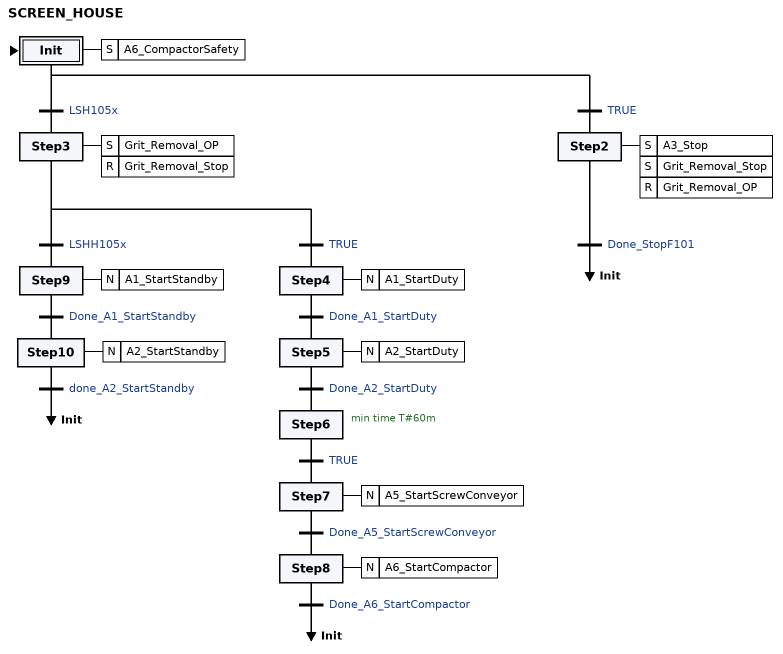
[picture p48: SCREEN_HOUSE (SFC)]
INITIAL_STEP Init:
	A6_CompactorSafety(S);
END_STEP
TRANSITION FROM Init TO Step3 := LSH105x;
END_TRANSITION
TRANSITION FROM Init TO Step2 := TRUE;
END_TRANSITION
STEP Step3:
	Grit_Removal_OP(S);
	Grit_Removal_Stop(R);
END_STEP
TRANSITION FROM Step3 TO Step9 := LSHH105x;
END_TRANSITION
TRANSITION FROM Step3 TO Step4 := TRUE;
END_TRANSITION
STEP Step9:
	A1_StartStandby(N);
END_STEP
TRANSITION FROM Step9 TO Step10 := Done_A1_StartStandby;
END_TRANSITION
STEP Step10:
	A2_StartStandby(N);
END_STEP
TRANSITION FROM Step10 TO Init := done_A2_StartStandby;
END_TRANSITION
STEP Step4:
	A1_StartDuty(N);
END_STEP
TRANSITION FROM Step4 TO Step5 := Done_A1_StartDuty;
END_TRANSITION
STEP Step5:
	A2_StartDuty(N);
END_STEP
TRANSITION FROM Step5 TO Step6 := Done_A2_StartDuty;
END_TRANSITION
STEP Step6: (* min time T#60m *)
END_STEP
TRANSITION FROM Step6 TO Step7 := TRUE;
END_TRANSITION
STEP Step7:
	A5_StartScrewConveyor(N);
END_STEP
TRANSITION FROM Step7 TO Step8 := Done_A5_StartScrewConveyor;
END_TRANSITION
STEP Step8:
	A6_StartCompactor(N);
END_STEP
TRANSITION FROM Step8 TO Init := Done_A6_StartCompactor;
END_TRANSITION
STEP Step2:
	A3_Stop(S);
	Grit_Removal_Stop(S);
	Grit_Removal_OP(R);
END_STEP
TRANSITION FROM Step2 TO Init := Done_StopF101;
END_TRANSITION
END_FUNCTION_BLOCK
ACTION A1_StartDuty:
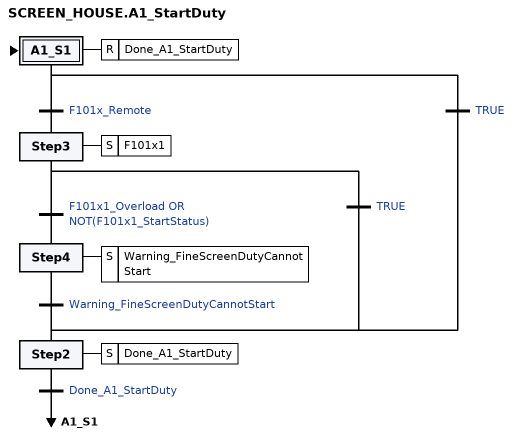
INITIAL_STEP A1_S1:
	Done_A1_StartDuty(R);
END_STEP
TRANSITION FROM A1_S1 TO Step3 := F101x_Remote;
END_TRANSITION
TRANSITION FROM A1_S1 TO Step2 := TRUE;
END_TRANSITION
STEP Step3:
	F101x1(S);
END_STEP
TRANSITION FROM Step3 TO Step4 := F101x1_Overload OR NOT(F101x1_StartStatus);
END_TRANSITION
TRANSITION FROM Step3 TO Step2 := TRUE;
END_TRANSITION
STEP Step4:
	Warning_FineScreenDutyCannotStart(S);
END_STEP
TRANSITION FROM Step4 TO Step2 := Warning_FineScreenDutyCannotStart;
END_TRANSITION
STEP Step2:
	Done_A1_StartDuty(S);
END_STEP
TRANSITION FROM Step2 TO A1_S1 := Done_A1_StartDuty;
END_TRANSITION
END_ACTION
ACTION A1_StartStandby:
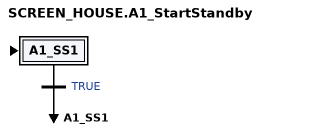
INITIAL_STEP A1_SS1:
END_STEP
TRANSITION FROM A1_SS1 TO A1_SS1 := TRUE;
END_TRANSITION
END_ACTION
ACTION A1_StopDuty:
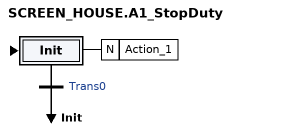
INITIAL_STEP Init:
	Action_1(N);
END_STEP
TRANSITION FROM Init TO Init := Trans0;
END_TRANSITION
END_ACTION
ACTION A1_StopStandby:
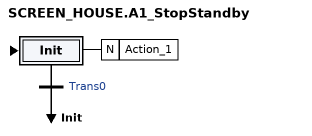
INITIAL_STEP Init:
	Action_1(N);
END_STEP
TRANSITION FROM Init TO Init := Trans0;
END_TRANSITION
END_ACTION
ACTION A2_StartDuty:
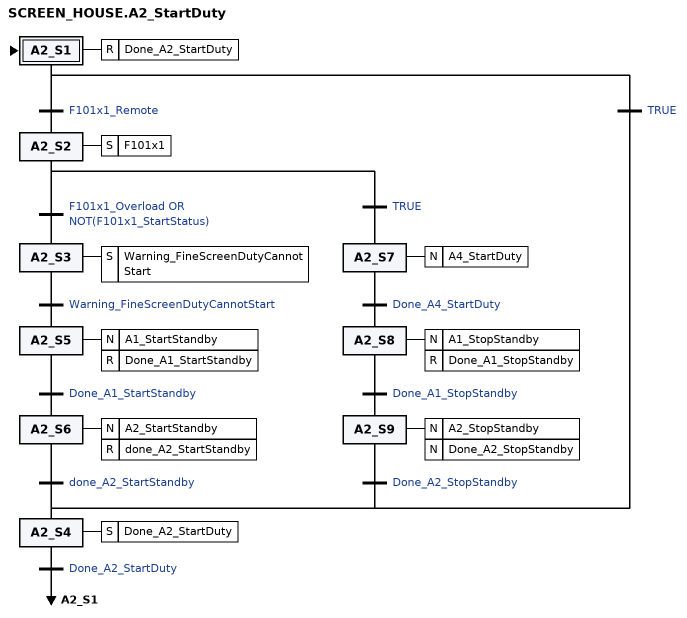
INITIAL_STEP A2_S1:
	Done_A2_StartDuty(R);
END_STEP
TRANSITION FROM A2_S1 TO A2_S2 := F101x1_Remote;
END_TRANSITION
TRANSITION FROM A2_S1 TO A2_S4 := TRUE;
END_TRANSITION
STEP A2_S2:
	F101x1(S);
END_STEP
TRANSITION FROM A2_S2 TO A2_S3 := F101x1_Overload OR NOT(F101x1_StartStatus);
END_TRANSITION
TRANSITION FROM A2_S2 TO A2_S7 := TRUE;
END_TRANSITION
STEP A2_S3:
	Warning_FineScreenDutyCannotStart(S);
END_STEP
TRANSITION FROM A2_S3 TO A2_S5 := Warning_FineScreenDutyCannotStart;
END_TRANSITION
STEP A2_S5:
	A1_StartStandby(N);
	Done_A1_StartStandby(R);
END_STEP
TRANSITION FROM A2_S5 TO A2_S6 := Done_A1_StartStandby;
END_TRANSITION
STEP A2_S6:
	A2_StartStandby(N);
	done_A2_StartStandby(R);
END_STEP
TRANSITION FROM A2_S6 TO A2_S4 := done_A2_StartStandby;
END_TRANSITION
STEP A2_S7:
	A4_StartDuty(N);
END_STEP
TRANSITION FROM A2_S7 TO A2_S8 := Done_A4_StartDuty;
END_TRANSITION
STEP A2_S8:
	A1_StopStandby(N);
	Done_A1_StopStandby(R);
END_STEP
TRANSITION FROM A2_S8 TO A2_S9 := Done_A1_StopStandby;
END_TRANSITION
STEP A2_S9:
	A2_StopStandby(N);
	Done_A2_StopStandby(N);
END_STEP
TRANSITION FROM A2_S9 TO A2_S4 := Done_A2_StopStandby;
END_TRANSITION
STEP A2_S4:
	Done_A2_StartDuty(S);
END_STEP
TRANSITION FROM A2_S4 TO A2_S1 := Done_A2_StartDuty;
END_TRANSITION
END_ACTION
ACTION A2_StartStandby:
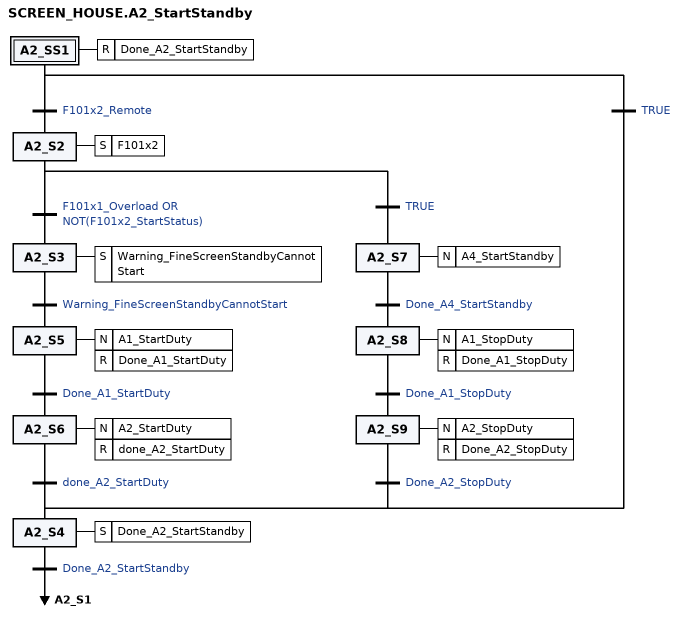
INITIAL_STEP A2_SS1:
	Done_A2_StartStandby(R);
END_STEP
TRANSITION FROM A2_SS1 TO A2_S2 := F101x2_Remote;
END_TRANSITION
TRANSITION FROM A2_SS1 TO A2_S4 := TRUE;
END_TRANSITION
STEP A2_S2:
	F101x2(S);
END_STEP
TRANSITION FROM A2_S2 TO A2_S3 := F101x1_Overload OR NOT(F101x2_StartStatus);
END_TRANSITION
TRANSITION FROM A2_S2 TO A2_S7 := TRUE;
END_TRANSITION
STEP A2_S3:
	Warning_FineScreenStandbyCannotStart(S);
END_STEP
TRANSITION FROM A2_S3 TO A2_S5 := Warning_FineScreenStandbyCannotStart;
END_TRANSITION
STEP A2_S5:
	A1_StartDuty(N);
	Done_A1_StartDuty(R);
END_STEP
TRANSITION FROM A2_S5 TO A2_S6 := Done_A1_StartDuty;
END_TRANSITION
STEP A2_S6:
	A2_StartDuty(N);
	done_A2_StartDuty(R);
END_STEP
TRANSITION FROM A2_S6 TO A2_S4 := done_A2_StartDuty;
END_TRANSITION
STEP A2_S7:
	A4_StartStandby(N);
END_STEP
TRANSITION FROM A2_S7 TO A2_S8 := Done_A4_StartStandby;
END_TRANSITION
STEP A2_S8:
	A1_StopDuty(N);
	Done_A1_StopDuty(R);
END_STEP
TRANSITION FROM A2_S8 TO A2_S9 := Done_A1_StopDuty;
END_TRANSITION
STEP A2_S9:
	A2_StopDuty(N);
	Done_A2_StopDuty(R);
END_STEP
TRANSITION FROM A2_S9 TO A2_S4 := Done_A2_StopDuty;
END_TRANSITION
STEP A2_S4:
	Done_A2_StartStandby(S);
END_STEP
TRANSITION FROM A2_S4 TO A2_S1 := Done_A2_StartStandby;
END_TRANSITION
END_ACTION
ACTION A2_StopDuty:
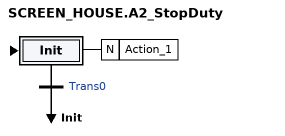
INITIAL_STEP Init:
	Action_1(N);
END_STEP
TRANSITION FROM Init TO Init := Trans0;
END_TRANSITION
END_ACTION
ACTION A2_StopStandby:
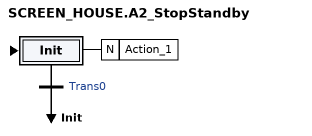
INITIAL_STEP Init:
	Action_1(N);
END_STEP
TRANSITION FROM Init TO Init := Trans0;
END_TRANSITION
END_ACTION
ACTION A3_Stop:
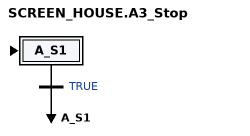
INITIAL_STEP A_S1:
END_STEP
TRANSITION FROM A_S1 TO A_S1 := TRUE;
END_TRANSITION
END_ACTION
ACTION A4_StartDuty:
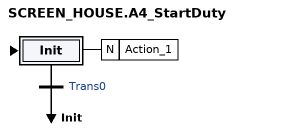
INITIAL_STEP Init:
	Action_1(N);
END_STEP
TRANSITION FROM Init TO Init := Trans0;
END_TRANSITION
END_ACTION
ACTION A4_StartStandby:
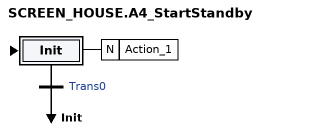
INITIAL_STEP Init:
	Action_1(N);
END_STEP
TRANSITION FROM Init TO Init := Trans0;
END_TRANSITION
END_ACTION
ACTION A5_ResetScrew:
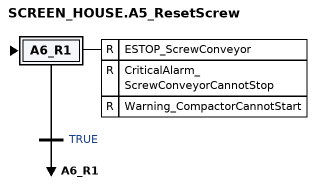
INITIAL_STEP A6_R1:
	ESTOP_ScrewConveyor(R);
	CriticalAlarm_ScrewConveyorCannotStop(R);
	Warning_CompactorCannotStart(R);
END_STEP
TRANSITION FROM A6_R1 TO A6_R1 := TRUE;
END_TRANSITION
END_ACTION
ACTION A5_StartScrewConveyor:
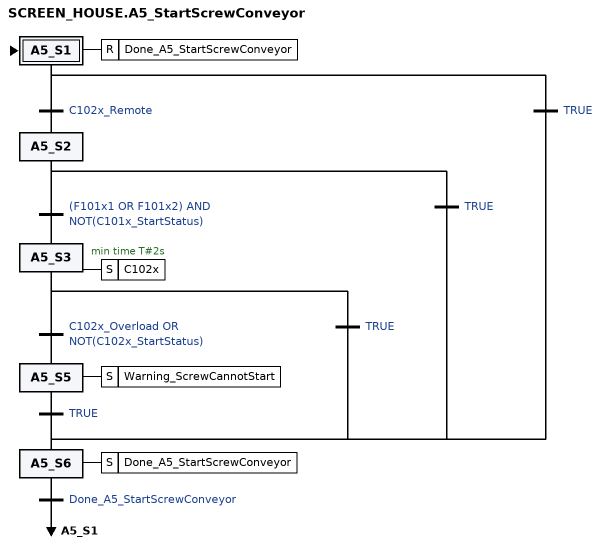
INITIAL_STEP A5_S1:
	Done_A5_StartScrewConveyor(R);
END_STEP
TRANSITION FROM A5_S1 TO A5_S2 := C102x_Remote;
END_TRANSITION
TRANSITION FROM A5_S1 TO A5_S6 := TRUE;
END_TRANSITION
STEP A5_S2:
END_STEP
TRANSITION FROM A5_S2 TO A5_S3 := (F101x1 OR F101x2) AND NOT(C101x_StartStatus);
END_TRANSITION
TRANSITION FROM A5_S2 TO A5_S6 := TRUE;
END_TRANSITION
STEP A5_S3: (* min time T#2s *)
	C102x(S);
END_STEP
TRANSITION FROM A5_S3 TO A5_S5 := C102x_Overload OR NOT(C102x_StartStatus);
END_TRANSITION
TRANSITION FROM A5_S3 TO A5_S6 := TRUE;
END_TRANSITION
STEP A5_S5:
	Warning_ScrewCannotStart(S);
END_STEP
TRANSITION FROM A5_S5 TO A5_S6 := TRUE;
END_TRANSITION
STEP A5_S6:
	Done_A5_StartScrewConveyor(S);
END_STEP
TRANSITION FROM A5_S6 TO A5_S1 := Done_A5_StartScrewConveyor;
END_TRANSITION
END_ACTION
ACTION A5_StopScrewConveyor:
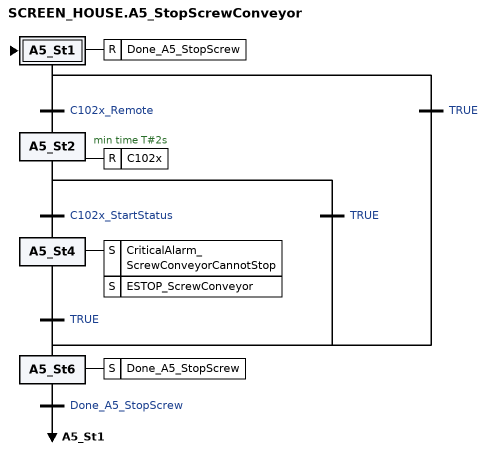
INITIAL_STEP A5_St1:
	Done_A5_StopScrew(R);
END_STEP
TRANSITION FROM A5_St1 TO A5_St2 := C102x_Remote;
END_TRANSITION
TRANSITION FROM A5_St1 TO A5_St6 := TRUE;
END_TRANSITION
STEP A5_St2: (* min time T#2s *)
	C102x(R);
END_STEP
TRANSITION FROM A5_St2 TO A5_St4 := C102x_StartStatus;
END_TRANSITION
TRANSITION FROM A5_St2 TO A5_St6 := TRUE;
END_TRANSITION
STEP A5_St4:
	CriticalAlarm_ScrewConveyorCannotStop(S);
	ESTOP_ScrewConveyor(S);
END_STEP
TRANSITION FROM A5_St4 TO A5_St6 := TRUE;
END_TRANSITION
STEP A5_St6:
	Done_A5_StopScrew(S);
END_STEP
TRANSITION FROM A5_St6 TO A5_St1 := Done_A5_StopScrew;
END_TRANSITION
END_ACTION
ACTION A6_CompactorSafety:
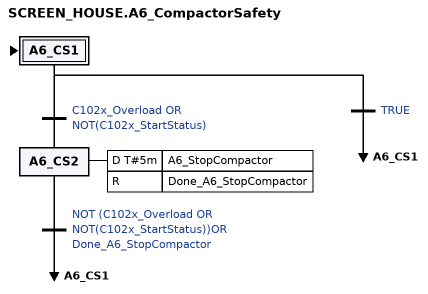
INITIAL_STEP A6_CS1:
END_STEP
TRANSITION FROM A6_CS1 TO A6_CS2 := C102x_Overload OR NOT(C102x_StartStatus);
END_TRANSITION
TRANSITION FROM A6_CS1 TO A6_CS1 := TRUE;
END_TRANSITION
STEP A6_CS2:
	A6_StopCompactor(D, T#5m);
	Done_A6_StopCompactor(R);
END_STEP
TRANSITION FROM A6_CS2 TO A6_CS1 := NOT (C102x_Overload OR NOT(C102x_StartStatus))OR Done_A6_StopCompactor;
END_TRANSITION
END_ACTION
ACTION A6_ResetCompactor:
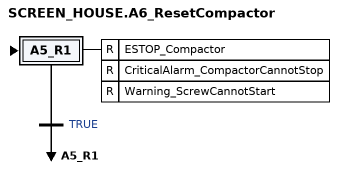
INITIAL_STEP A5_R1:
	ESTOP_Compactor(R);
	CriticalAlarm_CompactorCannotStop(R);
	Warning_ScrewCannotStart(R);
END_STEP
TRANSITION FROM A5_R1 TO A5_R1 := TRUE;
END_TRANSITION
END_ACTION
ACTION A6_StartCompactor:
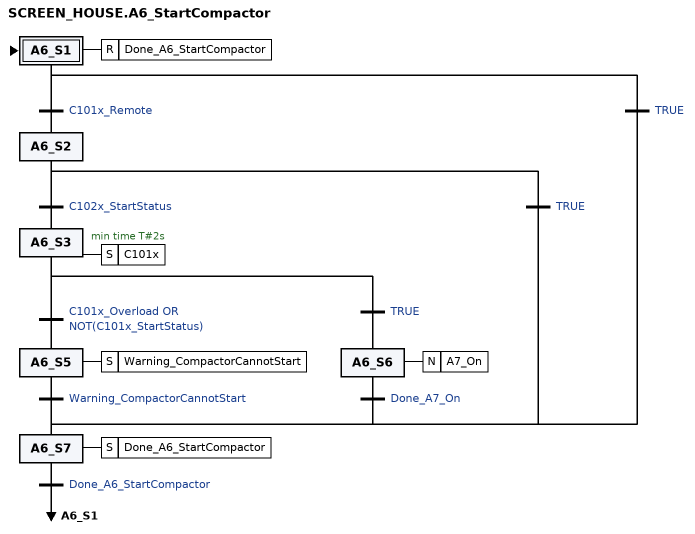
INITIAL_STEP A6_S1:
	Done_A6_StartCompactor(R);
END_STEP
TRANSITION FROM A6_S1 TO A6_S2 := C101x_Remote;
END_TRANSITION
TRANSITION FROM A6_S1 TO A6_S7 := TRUE;
END_TRANSITION
STEP A6_S2:
END_STEP
TRANSITION FROM A6_S2 TO A6_S3 := C102x_StartStatus;
END_TRANSITION
TRANSITION FROM A6_S2 TO A6_S7 := TRUE;
END_TRANSITION
STEP A6_S3: (* min time T#2s *)
	C101x(S);
END_STEP
TRANSITION FROM A6_S3 TO A6_S5 := C101x_Overload OR NOT(C101x_StartStatus);
END_TRANSITION
TRANSITION FROM A6_S3 TO A6_S6 := TRUE;
END_TRANSITION
STEP A6_S5:
	Warning_CompactorCannotStart(S);
END_STEP
TRANSITION FROM A6_S5 TO A6_S7 := Warning_CompactorCannotStart;
END_TRANSITION
STEP A6_S6:
	A7_On(N);
END_STEP
TRANSITION FROM A6_S6 TO A6_S7 := Done_A7_On;
END_TRANSITION
STEP A6_S7:
	Done_A6_StartCompactor(S);
END_STEP
TRANSITION FROM A6_S7 TO A6_S1 := Done_A6_StartCompactor;
END_TRANSITION
END_ACTION
ACTION A6_StopCompactor:
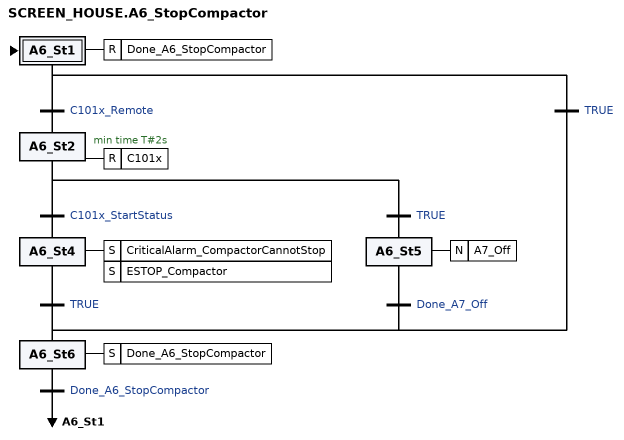
INITIAL_STEP A6_St1:
	Done_A6_StopCompactor(R);
END_STEP
TRANSITION FROM A6_St1 TO A6_St2 := C101x_Remote;
END_TRANSITION
TRANSITION FROM A6_St1 TO A6_St6 := TRUE;
END_TRANSITION
STEP A6_St2: (* min time T#2s *)
	C101x(R);
END_STEP
TRANSITION FROM A6_St2 TO A6_St4 := C101x_StartStatus;
END_TRANSITION
TRANSITION FROM A6_St2 TO A6_St5 := TRUE;
END_TRANSITION
STEP A6_St4:
	CriticalAlarm_CompactorCannotStop(S);
	ESTOP_Compactor(S);
END_STEP
TRANSITION FROM A6_St4 TO A6_St6 := TRUE;
END_TRANSITION
STEP A6_St5:
	A7_Off(N);
END_STEP
TRANSITION FROM A6_St5 TO A6_St6 := Done_A7_Off;
END_TRANSITION
STEP A6_St6:
	Done_A6_StopCompactor(S);
END_STEP
TRANSITION FROM A6_St6 TO A6_St1 := Done_A6_StopCompactor;
END_TRANSITION
END_ACTION
ACTION A7_Off:
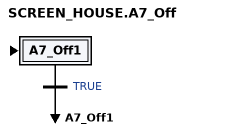
INITIAL_STEP A7_Off1:
END_STEP
TRANSITION FROM A7_Off1 TO A7_Off1 := TRUE;
END_TRANSITION
END_ACTION
ACTION A7_On:
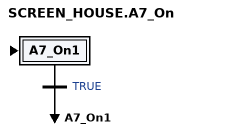
INITIAL_STEP A7_On1:
END_STEP
TRANSITION FROM A7_On1 TO A7_On1 := TRUE;
END_TRANSITION
END_ACTION
ACTION Grit_Removal_OP:
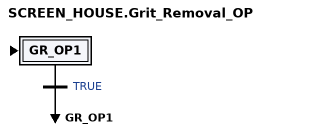
INITIAL_STEP GR_OP1:
END_STEP
TRANSITION FROM GR_OP1 TO GR_OP1 := TRUE;
END_TRANSITION
END_ACTION
ACTION Grit_Removal_Stop:
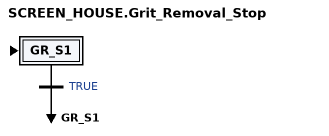
INITIAL_STEP GR_S1:
END_STEP
TRANSITION FROM GR_S1 TO GR_S1 := TRUE;
END_TRANSITION
END_ACTION
ACTION test:
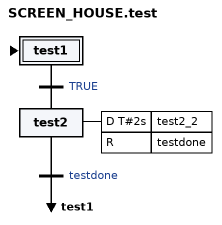
INITIAL_STEP test1:
END_STEP
TRANSITION FROM test1 TO test2 := TRUE;
END_TRANSITION
STEP test2:
	test2_2(D, T#2s);
	testdone(R);
END_STEP
TRANSITION FROM test2 TO test1 := testdone;
END_TRANSITION
END_ACTION
ACTION test2_2:
